// TIA Portal V21 export
VAR_GLOBAL   // PLC tag table "K_SegnaliMacchine"
END_VAR
VAR_GLOBAL CONSTANT   // user constants
   K_SegnaliMacchinaFasciatrice : Int := 12;
   K_SegnaliMacchinaPallettizzatore : Int := 11;
   K_SegnaliMacchinaFardellatrice : Int := 10;
   K_SegnaliMacchinaCluster : Int := 9;
   K_SegnaliMacchinaRaggiX : Int := 8;
   K_SegnaliMacchinaControlloVuoto : Int := 7;
   K_SegnaliMacchinaEtichettatrice : Int := 6;
   K_SegnaliMacchinaTrasporti : Int := 5;
   K_SegnaliMacchinaGruppoRiempi : Int := 4;
   K_SegnaliMacchinaDepal : Int := 3;
   K_SegnaliMacchinaPastorizzatore : Int := 2;
   K_SegnaliMacchinaTagTables : Int := 1;
   K_SegnaliMacchinaRobopackCFT : Int := 2;
   K_SegnaliMacchinaQCI : Int := 1;
END_VAR
